TYPE udtDBInterface :
STRUCT
	Trigger: DWORD;
	Response: DWORD;
	Lock: BOOL;
	Connection: ARRAY[0..19] OF udtDBChannel;
END_STRUCT
END_TYPE

(* stored: Version 1.1.0.1, ProductVersion 3.1.4020.12
   DUT udtDBInterface: Id {a0e75286-4de3-4bc4-bd8e-81bf56c76111} *)
